{attribute addProperty BoxType "EL2521-0124-0018"}
{attribute addProperty Id "ControlAT %Q*Control_055E5E7E1621Switch_on_valueAT %Q*UINT16217Switch_off_valueAT %Q*UINT16218"}
{attribute addProperty CRC "4159293044"}
{attribute addProperty SizeInBites "48"}
{attribute addProperty SizeInBytes "6"}
TYPE PLS_Control_compact_F7E9C674 :
STRUCT
	{attribute addProperty Name "Control"}
	Control AT %Q* : Control_055E5E7E;
	{attribute addProperty Name "Switch_on_value"}
	Switch_on_value AT %Q* : UINT;
	{attribute addProperty Name "Switch_off_value"}
	Switch_off_value AT %Q* : UINT;
END_STRUCT
END_TYPE

(* stored: Version 1.2.0.0, ProductVersion 3.1.4024.9
   DUT PLS_Control_compact_F7E9C674: Id {dc04c978-007f-4a3c-93cf-2ea83cdc8a01} *)
